INTERFACE I_ContinuousDrive EXTENDS I_Drive

METHOD ABSTRACT moveContinuous : BOOL
VAR_INPUT
	direction : MC_Direction;
END_VAR
END_METHOD

END_INTERFACE

(* stored: Version 1.1.0.1, ProductVersion 3.1.4024.11
   Itf I_ContinuousDrive: Id {80a1fc21-5f9a-49d6-a5a6-ad70aaa59166}
   Method moveContinuous: Id {077328e5-23f4-41ae-86eb-f7dd0288923b} *)
